FUNCTION_BLOCK INTERNAL FINAL FB_RoundTripDoubleTests EXTENDS FB_TestSuite
VAR CONSTANT
    cExpected : LREAL := 13.37000005;
END_VAR
VAR
    fbWriteCtx      : FB_WriteContext;
    fbParseCtx      : FB_ParseContext;
    aBuffer         : ARRAY[0..15] OF BYTE;
    hrWriterActual  : HRESULT;
    hrParserActual  : HRESULT;
    fActual         : LREAL;
END_VAR

TEST(__POUNAME());

// Arrange
fbWriteCtx.FromBuffer(aBuffer);
fbWriteCtx.refCtx.stState.nBufferPos := 2;
fbParseCtx.FromBuffer(aBuffer);
fbParseCtx.refCtx.stState.nBufferPos := 2;

// Act
hrWriterActual := F_WriteDouble(fbWriteCtx.refCtx, cExpected);
hrParserActual := F_ParseDouble(fbParseCtx.refCtx, fVAlue=> fActual);

// Assert
AssertEquals_DINT(Expected:= S_OK, Actual:= hrWriterActual, Message:= 'Expected hrWriterActual = S_OK');
AssertEquals_DINT(Expected:= S_OK, Actual:= hrParserActual, Message:= 'Expected hrParserActual = S_OK');
AssertEquals_LREAL(Expected:= cExpected, Actual:= fActual, Delta:= 4.94065645841247E-324, Message:= 'Values differ');

TEST_FINISHED_NAMED(__POUNAME());

END_FUNCTION_BLOCK

(* stored: Version 1.1.0.1
   POU FB_RoundTripDoubleTests: Id {70f5849c-d2c6-4a04-ba24-4d36a927c042}, SpecialFunc None *)
